// TIA Portal V18 export
DATA_BLOCK "TD_Control_DB"   // DB19
// stored: AutoNumber false, InstanceOfName TD_Control, InstanceOfType FB
"TD_Control"
   // VAR
   //    AllowShift : Bool;
   //    TD_Mode : Int;
   //    HSLTShift_TP { S7_SetPoint := 'True'} : TP_TIME;
   //    LSHTShift_TP { S7_SetPoint := 'True'} : TP_TIME;
   //    MUSpinComplete : Bool;
   //    TDP1FwdSetmA : Real;
   //    TDP2FwdSetmA : Real;
   //    TDP1RevSetmA : Real;
   //    TDP2RevSetmA : Real;
   //    TorqSetmA : Real;
   //    TDP1FwdEn : Bool;
   //    TDP2FwdEn : Bool;
   //    TDP1RevEn : Bool;
   //    TDP2RevEn : Bool;
   //    TorqEn : Bool;
   //    BypassDelay_TON { S7_SetPoint := 'True'} : TON_TIME;
   //    BypassRunning_TOF { S7_SetPoint := 'True'} : TOF_TIME;
   //    HSLT_Sol_Last { S7_SetPoint := 'True'} : Bool;
   //    LSHT_Sol_Last : Bool;
   //    AllowRev : Bool;
   //    SpeedLimiting : Bool;
   //    SpeedLimitmAOut : Real;
   //    SpeedLimitingTrig : Bool;
   //    MUTorqStart : Bool;
   //    BOStart : Bool;
   //    OscStart : Bool;
   //    MUTorqStart_Trig : Bool;
   //    BOStart_Trig : Bool;
   //    OscStart_Trig : Bool;
   //    SpeedLimit_SlewDec { S7_SetPoint := 'True'} : "SlewDec";
   //    SpeedLimit_SlewInc { S7_SetPoint := 'True'} : "SlewInc";
   //    HiTempShutDown_TON { S7_SetPoint := 'True'} : TON_TIME;
   // END_VAR
BEGIN
END_DATA_BLOCK
